(* PLC project  *)

PROGRAM P

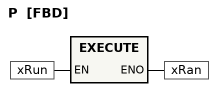
(* FBD diagram, written out as Structured Text *)
IF xRun THEN
  a := 1;
  b := 2;
END_IF;
xRan := xRun;
END_PROGRAM
